FUNCTION_BLOCK WriteBoolIf
VAR_IN_OUT
	Out: BOOL;
END_VAR
VAR_INPUT
	EN: BOOL := TRUE;
	In: BOOL;
END_VAR
VAR_OUTPUT
	ENO: BOOL;
END_VAR
VAR
END_VAR

ENO := EN;
IF EN THEN
	Out := In;
END_IF

END_FUNCTION_BLOCK

(* stored: Version 1.1.0.1, ProductVersion 3.1.4024.5
   POU WriteBoolIf: Id {e1d5238b-e53c-4fdc-ae3a-44a96228925f}, SpecialFunc None *)
